(* CoDeSys 2.3 export: PLC_PRG.EXP *)

(* POU PLC_PRG, FBD *)
PROGRAM PLC_PRG
VAR
	Init1: BOOL:=TRUE;
	CycleTime:DWORD;
	MaxCycleTime:DWORD;
	ResetMax:BOOL;
END_VAR
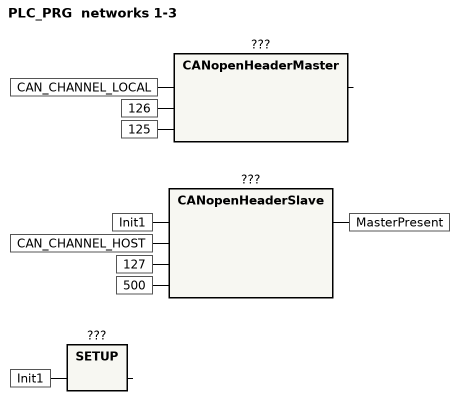
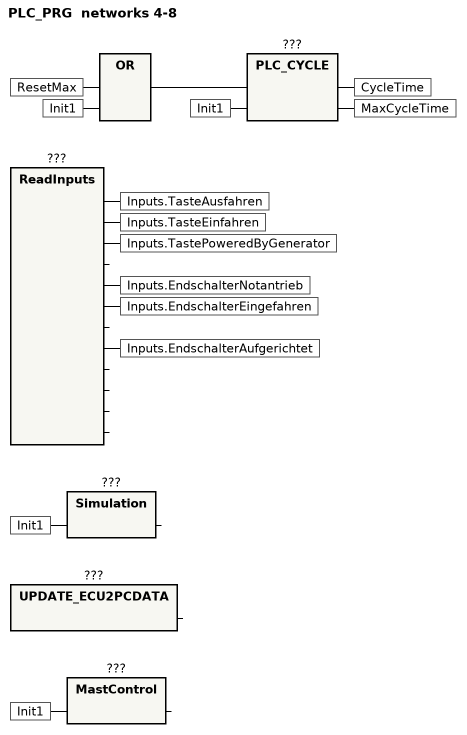
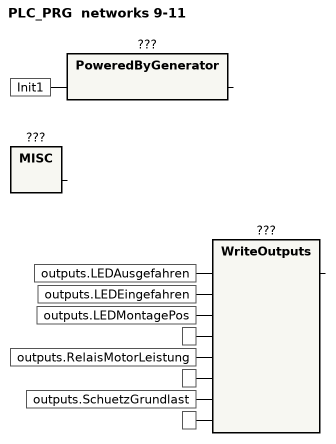
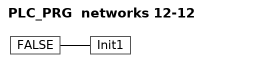
_FBD_ (* Function Block Diagram *)
NETWORK 1 (* CAN Master auf CAN2 initialisieren (Schnittstelle zu FU) *)
	???:CANopenHeaderMaster(CAN_CHANNEL_LOCAL, 126, 125)
NETWORK 2 (* CAN Slave auf CAN1 initialisieren (Schnittstelle zu PC) *)
	???:CANopenHeaderSlave(Init1, CAN_CHANNEL_HOST, 127, 500) => MasterPresent
NETWORK 3
	???:SETUP(Init1)
NETWORK 4
	???:PLC_CYCLE(OR(ResetMax, Init1), Init1, out 2 => MaxCycleTime) => CycleTime
NETWORK 5
	???:ReadInputs(out 2 => Inputs.TasteEinfahren, out 3 => Inputs.TastePoweredByGenerator, out 5 => Inputs.EndschalterNotantrieb, out 6 => Inputs.EndschalterEingefahren, out 8 => Inputs.EndschalterAufgerichtet) => Inputs.TasteAusfahren
NETWORK 6
	???:Simulation(Init1)
NETWORK 7
	???:UPDATE_ECU2PCDATA()
NETWORK 8
	NOT ???:MastControl(Init1)
NETWORK 9
	???:PoweredByGenerator(Init1)
NETWORK 10
	???:MISC()
NETWORK 11
	???:WriteOutputs(outputs.LEDAusgefahren, outputs.LEDEingefahren, outputs.LEDMontagePos, , outputs.RelaisMotorLeistung, , outputs.SchuetzGrundlast, )
NETWORK 12 (* last line *)
	FALSE => Init1
_END_FBD_
(* the same logic as Structured Text *)
(* Network 1: see the listing above *)
(* Network 2: see the listing above *)
(* Network 3: see the listing above *)
(* Network 4: see the listing above *)
(* Network 5: see the listing above *)
(* Network 6: see the listing above *)
(* Network 7: see the listing above *)
(* Network 8: see the listing above *)
(* Network 9: see the listing above *)
(* Network 10: see the listing above *)
(* Network 11: see the listing above *)
(* Network 12 *)
Init1 := FALSE;
END_PROGRAM
